{attribute 'reflection'}
FUNCTION_BLOCK Derivative IMPLEMENTS IOut
VAR_INPUT
    value : LREAL;
    deltaTime : Millisecond;
END_VAR
VAR
    {attribute 'instance-path'}
    {attribute 'noinit'}
    _path : Tc2_System.T_MaxString;
    _out : LREAL;
    _previousValue : LREAL;
    _firstCall : BOOL := TRUE;
END_VAR

IF _firstCall THEN
    _firstCall := FALSE;
ELSE
    IF deltaTime <> 0 THEN
        _out := (value - _previousValue) / deltaTime;
    ELSE
        ADSLOGSTR(
            msgCtrlMask:=ADSLOG_MSGTYPE_ERROR,
            msgFmtStr:='%s: Enter a delta time > 0!',
            strArg:=_path
        );
    END_IF
END_IF
_previousValue := value;

PROPERTY Out : LREAL
GET
Out := _out;
END_GET
END_PROPERTY

END_FUNCTION_BLOCK

(* stored: Version 1.1.0.1, ProductVersion 3.1.4024.12
   POU Derivative: Id {c4c45863-dcb9-41dd-861c-a4ff025142ae}, SpecialFunc None
   Property Out: Id {a6db672b-0b34-404c-9e80-4de00c4fcb64}
   Get Get: Id {d27e6734-47dd-49be-9122-f5b93be0d613} *)
